TYPE MultiAxis_Input_typ :
	STRUCT
		Command 	: MultiAxis_CMD_typ ;
		Parameter	: MultiAxis_Param_typ ;
	END_STRUCT
END_TYPE

(* stored: Version 1.1.0.1, ProductVersion 3.1.4024.3
   DUT MultiAxis_Input_typ: Id {36ff22db-3c76-0410-23e0-a5cbfa5f5321} *)
